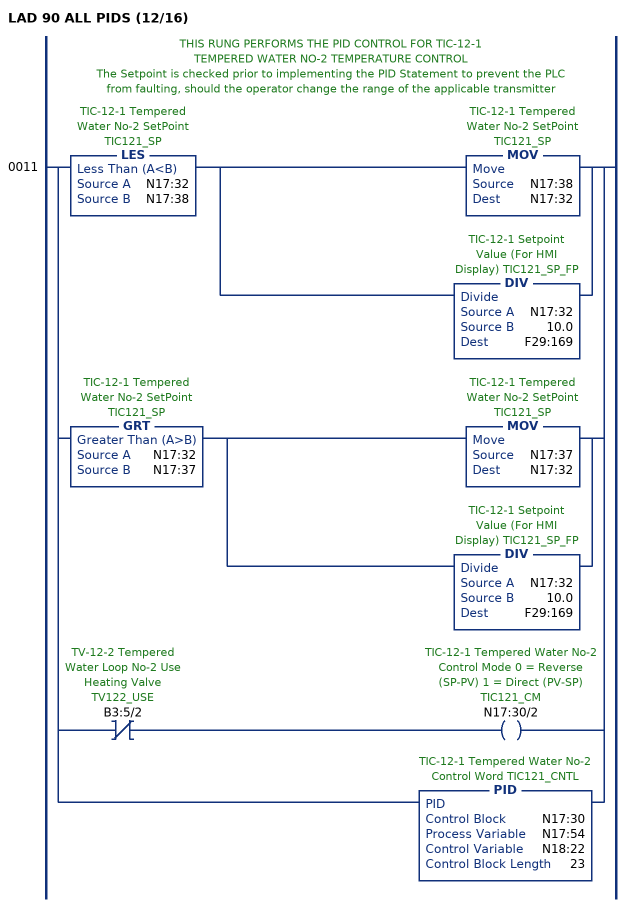
% Rung: 11 %
% THIS RUNG PERFORMS THE PID CONTROL FOR TIC-12-1
% TEMPERED WATER NO-2 TEMPERATURE CONTROL
% The Setpoint is checked prior to implementing the PID Statement to prevent the PLC
% from faulting, should the operator change the range of the applicable transmitter %
SOR BST LES N17:32 N17:38 BST MOV N17:38 N17:32 NXB DIV N17:32 10.0 F29:169 BND NXB GRT N17:32 N17:37 BST MOV N17:37 N17:32 NXB DIV N17:32 10.0 F29:169 BND NXB XIO B3:5/2 OTE N17:30/2 NXB PID N17:30 N17:54 N18:22 23 BND EOR
%   N17:32  TIC121_SP  "TIC-12-1 Tempered Water No-2 SetPoint" %
%   N17:38  TIC121_SMIN  "TIC-12-1 Tempered Water No-2 Setpoint Minimum" %
%   F29:169  TIC121_SP_FP  "TIC-12-1 Setpoint Value (For HMI Display)" %
%   N17:37  TIC121_SMAX  "TIC-12-1 Tempered Water No-2 Setpoint Maximum" %
%   B3:5/2  TV122_USE  "TV-12-2 Tempered Water Loop No-2 Use Heating Valve" %
%   N17:30/2  TIC121_CM  "TIC-12-1 Tempered Water No-2 Control Mode 0 = Reverse (SP-PV) 1 = Direct (PV-SP)" %
%   N17:30  TIC121_CNTL  "TIC-12-1 Tempered Water No-2 Control Word" %
%   N17:54  TIC121_IN  "TIC-12-1 Tempered Water No-2 Scaled Input" %
%   N18:22  TIC121_OUT1  "TIC-12-1 Tempered Water No-2 PID Output Value" %

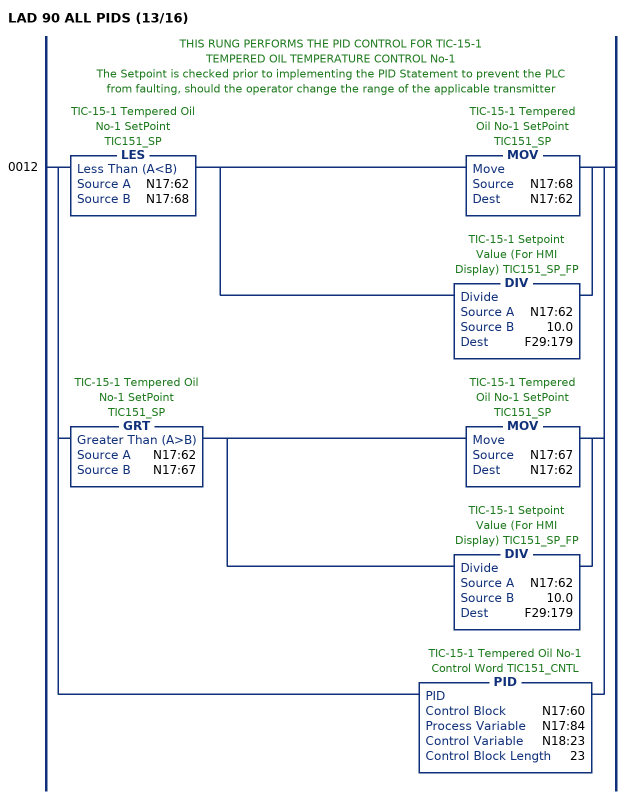
% Rung: 12 %
% THIS RUNG PERFORMS THE PID CONTROL FOR TIC-15-1
% TEMPERED OIL TEMPERATURE CONTROL No-1
% The Setpoint is checked prior to implementing the PID Statement to prevent the PLC
% from faulting, should the operator change the range of the applicable transmitter %
SOR BST LES N17:62 N17:68 BST MOV N17:68 N17:62 NXB DIV N17:62 10.0 F29:179 BND NXB GRT N17:62 N17:67 BST MOV N17:67 N17:62 NXB DIV N17:62 10.0 F29:179 BND NXB PID N17:60 N17:84 N18:23 23 BND EOR
%   N17:62  TIC151_SP  "TIC-15-1 Tempered Oil No-1 SetPoint" %
%   N17:68  TIC151_SMIN  "TIC-15-1 Tempered Oil No-1 Setpoint Minimum" %
%   F29:179  TIC151_SP_FP  "TIC-15-1 Setpoint Value (For HMI Display)" %
%   N17:67  TIC151_SMAX  "TIC-15-1 Tempered Oil No-1 Setpoint Maximum" %
%   N17:60  TIC151_CNTL  "TIC-15-1 Tempered Oil No-1 Control Word" %
%   N17:84  TIC151_IN  "TIC-15-1 Tempered Oil No-1 Scaled Input" %
%   N18:23  TIC151_OUT1  "TIC-15-1 Tempered Oil No-1 PID Output Value" %

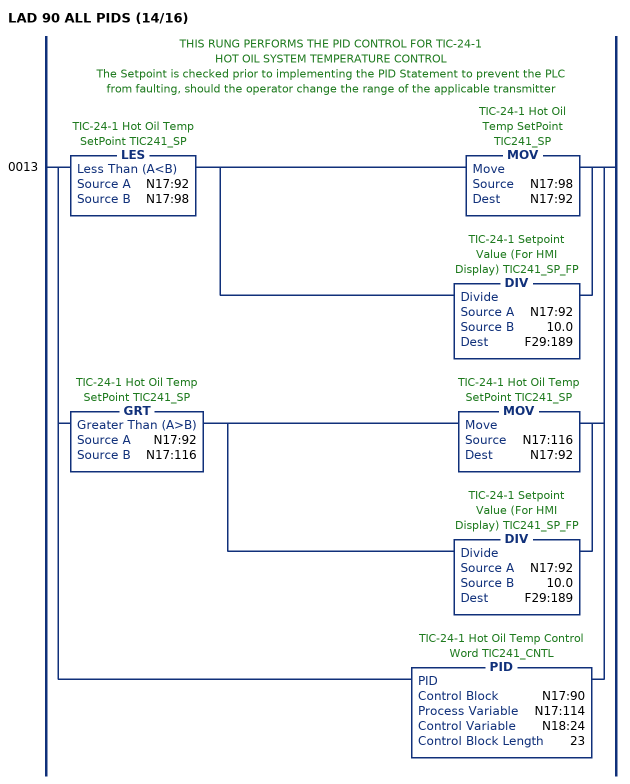
% Rung: 13 %
% THIS RUNG PERFORMS THE PID CONTROL FOR TIC-24-1
% HOT OIL SYSTEM TEMPERATURE CONTROL
% The Setpoint is checked prior to implementing the PID Statement to prevent the PLC
% from faulting, should the operator change the range of the applicable transmitter %
SOR BST LES N17:92 N17:98 BST MOV N17:98 N17:92 NXB DIV N17:92 10.0 F29:189 BND NXB GRT N17:92 N17:116 BST MOV N17:116 N17:92 NXB DIV N17:92 10.0 F29:189 BND NXB PID N17:90 N17:114 N18:24 23 BND EOR
%   N17:92  TIC241_SP  "TIC-24-1 Hot Oil Temp SetPoint" %
%   N17:98  TIC241_SMIN  "TIC-24-1 Hot Oil Temp Setpoint Minimum" %
%   F29:189  TIC241_SP_FP  "TIC-24-1 Setpoint Value (For HMI Display)" %
%   N17:116  TIC241_OPER_SPMAX  "TIC-24-1 Operating Setpoint Max" %
%   N17:90  TIC241_CNTL  "TIC-24-1 Hot Oil Temp Control Word" %
%   N17:114  TIC241_IN  "TIC-24-1 Hot Oil Temp Scaled Input" %
%   N18:24  TIC241_OUT1  "TIC-24-1 Hot Oil Temp PID Output Value" %

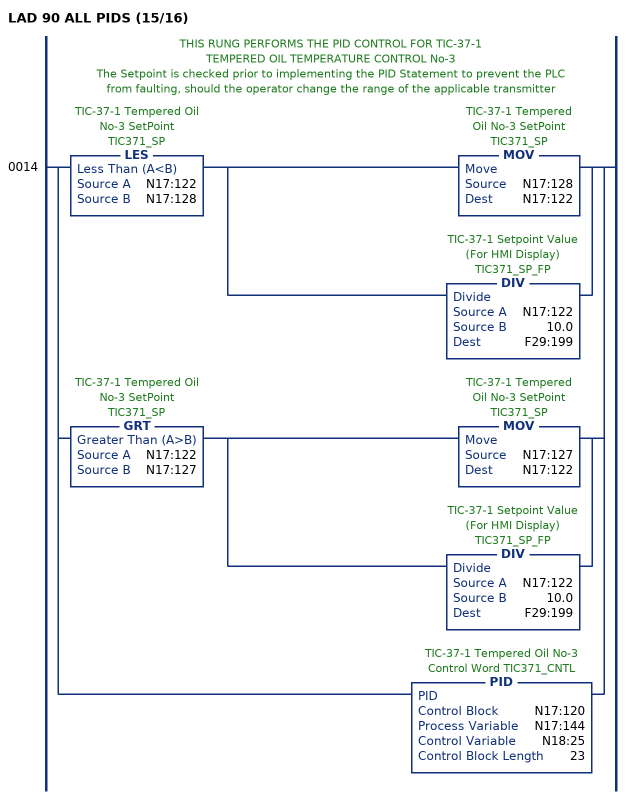
% Rung: 14 %
% THIS RUNG PERFORMS THE PID CONTROL FOR TIC-37-1
% TEMPERED OIL TEMPERATURE CONTROL No-3
% The Setpoint is checked prior to implementing the PID Statement to prevent the PLC
% from faulting, should the operator change the range of the applicable transmitter %
SOR BST LES N17:122 N17:128 BST MOV N17:128 N17:122 NXB DIV N17:122 10.0 F29:199 BND NXB GRT N17:122 N17:127 BST MOV N17:127 N17:122 NXB DIV N17:122 10.0 F29:199 BND NXB PID N17:120 N17:144 N18:25 23 BND EOR
%   N17:122  TIC371_SP  "TIC-37-1 Tempered Oil No-3 SetPoint" %
%   N17:128  TIC371_SMIN  "TIC-37-1 Tempered Oil No-3 Setpoint Minimum" %
%   F29:199  TIC371_SP_FP  "TIC-37-1 Setpoint Value (For HMI Display)" %
%   N17:127  TIC371_SMAX  "TIC-37-1 Tempered Oil No-3 Setpoint Maximum" %
%   N17:120  TIC371_CNTL  "TIC-37-1 Tempered Oil No-3 Control Word" %
%   N17:144  TIC371_IN  "TIC-37-1 Tempered Oil No-3 Scaled Input" %
%   N18:25  TIC371_OUT1  "TIC-37-1 Tempered Oil No-3 PID Output Value" %

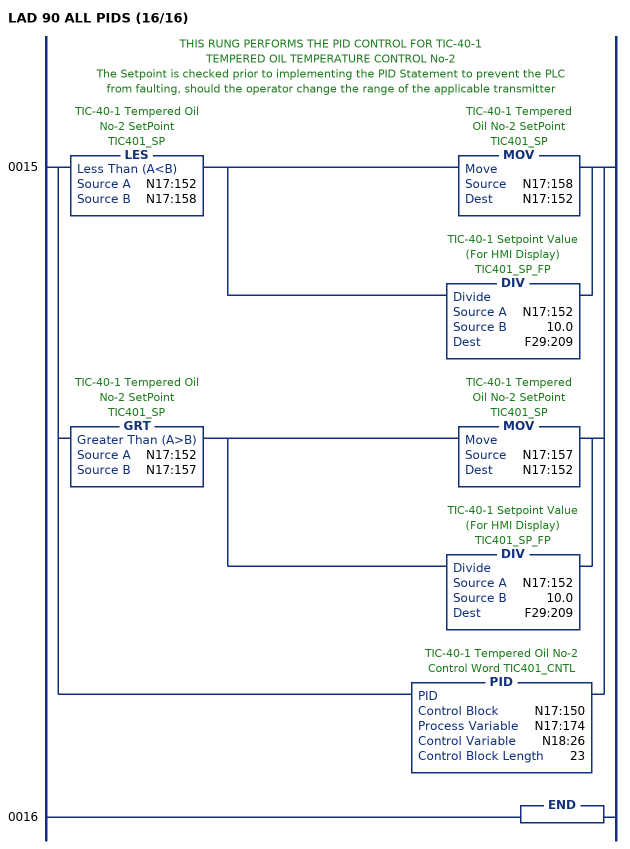
% Rung: 15 %
% THIS RUNG PERFORMS THE PID CONTROL FOR TIC-40-1
% TEMPERED OIL TEMPERATURE CONTROL No-2
% The Setpoint is checked prior to implementing the PID Statement to prevent the PLC
% from faulting, should the operator change the range of the applicable transmitter %
SOR BST LES N17:152 N17:158 BST MOV N17:158 N17:152 NXB DIV N17:152 10.0 F29:209 BND NXB GRT N17:152 N17:157 BST MOV N17:157 N17:152 NXB DIV N17:152 10.0 F29:209 BND NXB PID N17:150 N17:174 N18:26 23 BND EOR
%   N17:152  TIC401_SP  "TIC-40-1 Tempered Oil No-2 SetPoint" %
%   N17:158  TIC401_SMIN  "TIC-40-1 Tempered Oil No-2 Setpoint Minimum" %
%   F29:209  TIC401_SP_FP  "TIC-40-1 Setpoint Value (For HMI Display)" %
%   N17:157  TIC401_SMAX  "TIC-40-1 Tempered Oil No-2 Setpoint Maximum" %
%   N17:150  TIC401_CNTL  "TIC-40-1 Tempered Oil No-2 Control Word" %
%   N17:174  TIC401_IN  "TIC-40-1 Tempered Oil No-2 Scaled Input" %
%   N18:26  TIC401_OUT1  "TIC-40-1 Tempered Oil No-2 PID Output Value" %
% Rung: 16 %
SOR END EOR

LADDER 101 "FIC-21-1"    % Feed Flow No-1 PID Controls %
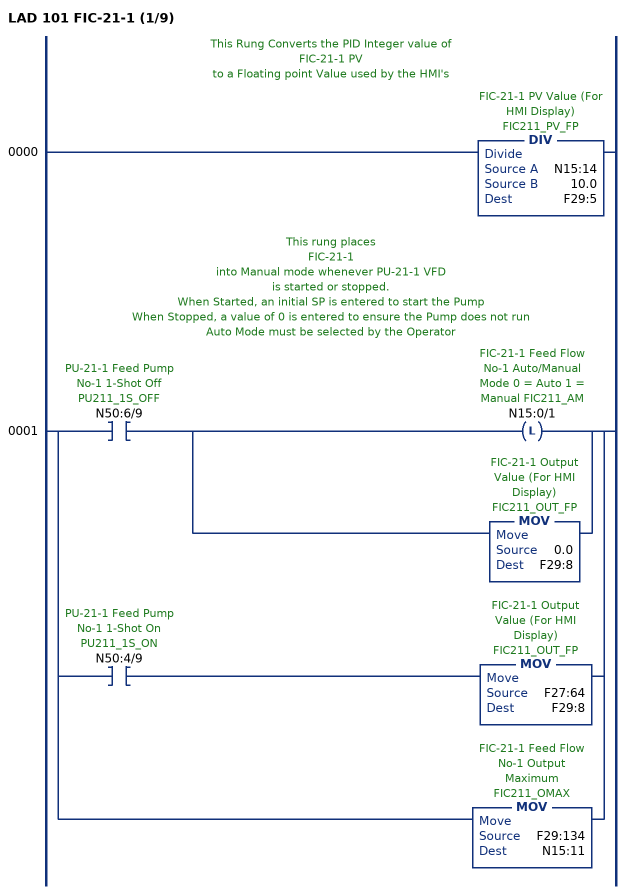
% Rung: 0 %
% This Rung Converts the PID Integer value of
% FIC-21-1 PV
% to a Floating point Value used by the HMI's %
SOR DIV N15:14 10.0 F29:5 EOR
%   N15:14  FIC211_PV  "FIC-21-1 Feed Flow No-1 Scaled Process Variable" %
%   F29:5  FIC211_PV_FP  "FIC-21-1 PV Value (For HMI Display)" %
% Rung: 1 %
% This rung places
% FIC-21-1
% into Manual mode whenever PU-21-1 VFD
% is started or stopped.
% When Started, an initial SP is entered to start the Pump
% When Stopped, a value of 0 is entered to ensure the Pump does not run
% Auto Mode must be selected by the Operator %
SOR BST XIC N50:6/9 BST OTL N15:0/1 NXB MOV 0.0 F29:8 BND NXB XIC N50:4/9 MOV F27:64 F29:8 NXB MOV F29:134 N15:11 BND EOR
%   N50:6/9  PU211_1S_OFF  "PU-21-1 Feed Pump No-1 1-Shot Off" %
%   N15:0/1  FIC211_AM  "FIC-21-1 Feed Flow No-1 Auto/Manual Mode 0 = Auto 1 = Manual" %
%   F29:8  FIC211_OUT_FP  "FIC-21-1 Output Value (For HMI Display)" %
%   N50:4/9  PU211_1S_ON  "PU-21-1 Feed Pump No-1 1-Shot On" %
%   F27:64  SIC211_INIT_SP  "SIC-21-1 Initial Speed Setpoint (Hz)" %
%   F29:134  SIC211_MAX  "SIC-21-1 PU-21-1 Feed Pump No-1 Freq at 100% Value (For HMI Display)" %
%   N15:11  FIC211_OMAX  "FIC-21-1 Feed Flow No-1 Output Maximum" %

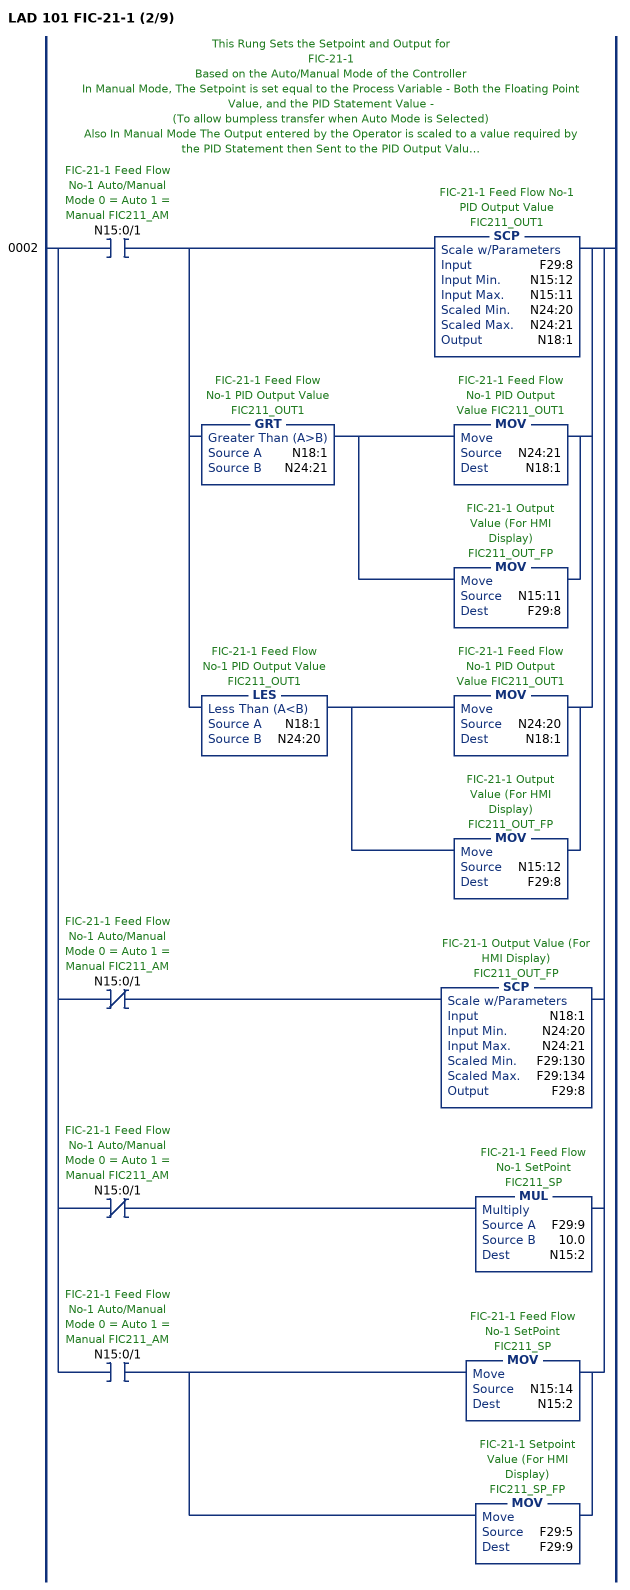
% Rung: 2 %
% This Rung Sets the Setpoint and Output for
% FIC-21-1
% Based on the Auto/Manual Mode of the Controller
% In Manual Mode, The Setpoint is set equal to the Process Variable - Both the Floating Point Value, and the PID Statement Value -
% (To allow bumpless transfer when Auto Mode is Selected)
% Also In Manual Mode The Output entered by the Operator is scaled to a value required by the PID Statement then Sent to the PID Output Value
% 
% In Auto Mode, The Setpoint is Entered by the Operator from Any HMI terminal, Multiplied by 10, and placed in the PID Statement's Setpoint Location
% Also In Auto Mode, the Output (used by the Operator) is set equal to the actual value of the pID statement
% (To allow bumpless transfer when Manual Mode is Selected) %
SOR BST XIC N15:0/1 BST SCP F29:8 N15:12 N15:11 N24:20 N24:21 N18:1 NXB GRT N18:1 N24:21 BST MOV N24:21 N18:1 NXB MOV N15:11 F29:8 BND NXB LES N18:1 N24:20 BST MOV N24:20 N18:1 NXB MOV N15:12 F29:8 BND BND NXB XIO N15:0/1 SCP N18:1 N24:20 N24:21 F29:130 F29:134 F29:8 NXB XIO N15:0/1 MUL F29:9 10.0 N15:2 NXB XIC N15:0/1 BST MOV N15:14 N15:2 NXB MOV F29:5 F29:9 BND BND EOR
%   N15:0/1  FIC211_AM  "FIC-21-1 Feed Flow No-1 Auto/Manual Mode 0 = Auto 1 = Manual" %
%   F29:8  FIC211_OUT_FP  "FIC-21-1 Output Value (For HMI Display)" %
%   N15:12  FIC211_OMIN  "FIC-21-1 Feed Flow No-1 Output Minimum" %
%   N15:11  FIC211_OMAX  "FIC-21-1 Feed Flow No-1 Output Maximum" %
%   N24:20  PID_MIN  "PID Statement Minimum Value" %
%   N24:21  PID_MAX  "PID Statement Maximum Value" %
%   N18:1  FIC211_OUT1  "FIC-21-1 Feed Flow No-1 PID Output Value" %
%   F29:130  SIC211_MIN  "SIC-21-1 PU-21-1 Feed Pump No-1 Speed 0% Value (For HMI Display)" %
%   F29:134  SIC211_MAX  "SIC-21-1 PU-21-1 Feed Pump No-1 Freq at 100% Value (For HMI Display)" %
%   F29:9  FIC211_SP_FP  "FIC-21-1 Setpoint Value (For HMI Display)" %
%   N15:2  FIC211_SP  "FIC-21-1 Feed Flow No-1 SetPoint" %
%   N15:14  FIC211_PV  "FIC-21-1 Feed Flow No-1 Scaled Process Variable" %
%   F29:5  FIC211_PV_FP  "FIC-21-1 PV Value (For HMI Display)" %

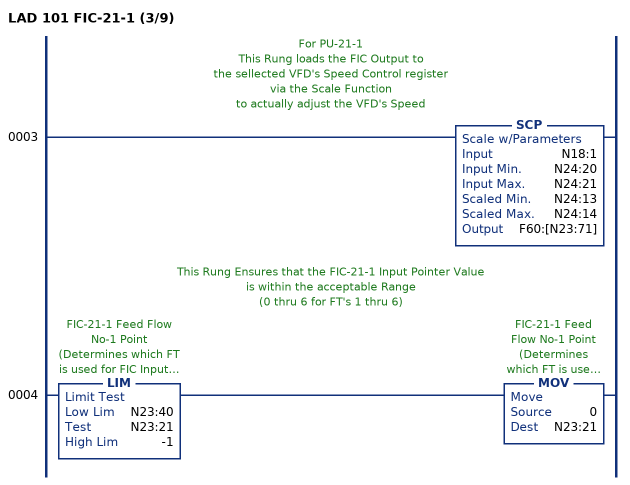
% Rung: 3 %
% For PU-21-1
% This Rung loads the FIC Output to
% the sellected VFD's Speed Control register
% via the Scale Function
% to actually adjust the VFD's Speed %
SOR SCP N18:1 N24:20 N24:21 N24:13 N24:14 F60:[N23:71] EOR
%   N18:1  FIC211_OUT1  "FIC-21-1 Feed Flow No-1 PID Output Value" %
%   N24:20  PID_MIN  "PID Statement Minimum Value" %
%   N24:21  PID_MAX  "PID Statement Maximum Value" %
%   N24:13  AO_MIN_OE4  "Analog Output Minimum Value Generates 4 mA DC (To OE4 AO Module)" %
%   N24:14  AO_MAX_OE4  "Analog Output Maximum Value Generates 20 mA DC (To OE4 AO Module)" %
%   N23:71  FIC211_OUT_PTR  "FIC-21-1 Feed Flow No-1 Output Pointer Determines which VFD is controled by FIC" %
% Rung: 4 %
% This Rung Ensures that the FIC-21-1 Input Pointer Value
% is within the acceptable Range
% (0 thru 6 for FT's 1 thru 6) %
SOR LIM N23:40 N23:21 -1 MOV 0 N23:21 EOR
%   N23:40  MAX_FT_ALLOWED_1  "Maximum Number of FTs Available Plus 1" %
%   N23:21  FIC211_IN_PTR  "FIC-21-1 Feed Flow No-1 Point (Determines which FT is used for FIC Input)" %

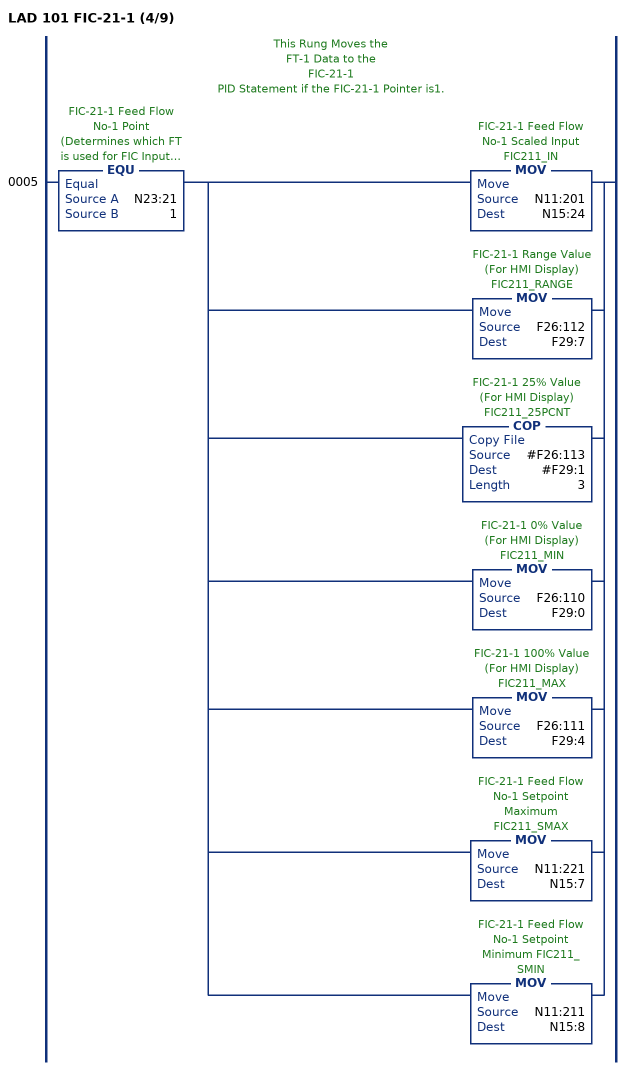
% Rung: 5 %
% This Rung Moves the
% FT-1 Data to the
% FIC-21-1
% PID Statement if the FIC-21-1 Pointer is1. %
SOR EQU N23:21 1 BST MOV N11:201 N15:24 NXB MOV F26:112 F29:7 NXB COP #F26:113 #F29:1 3 NXB MOV F26:110 F29:0 NXB MOV F26:111 F29:4 NXB MOV N11:221 N15:7 NXB MOV N11:211 N15:8 BND EOR
%   N23:21  FIC211_IN_PTR  "FIC-21-1 Feed Flow No-1 Point (Determines which FT is used for FIC Input)" %
%   N11:201  FT01_PID_IN  "FT-1 Flow Transmitter No-1 PID Statement Input Value" %
%   N15:24  FIC211_IN  "FIC-21-1 Feed Flow No-1 Scaled Input" %
%   F26:112  FT01_RANGE  "FT-1 Range Value (Max-Min)" %
%   F29:7  FIC211_RANGE  "FIC-21-1 Range Value (For HMI Display)" %
%   F26:113  FT01_25PCNT_VALUE  "FT-1 25% Range Value For HMI Display" %
%   F29:1  FIC211_25PCNT  "FIC-21-1 25% Value (For HMI Display)" %
%   F26:110  FT01_MIN  "FT-1 Minimum Value" %
%   F29:0  FIC211_MIN  "FIC-21-1 0% Value (For HMI Display)" %
%   F26:111  FT01_MAX  "FT-1 Maximum Value" %
%   F29:4  FIC211_MAX  "FIC-21-1 100% Value (For HMI Display)" %
%   N11:221  FT01_PID_MAX  "FT-1 Flow Transmitter No-1 PID Statement Maximum Input Value" %
%   N15:7  FIC211_SMAX  "FIC-21-1 Feed Flow No-1 Setpoint Maximum" %
%   N11:211  FT01_PID_MIN  "FT-1 Flow Transmitter No-1 PID Statement Minimum Input Value" %
%   N15:8  FIC211_SMIN  "FIC-21-1 Feed Flow No-1 Setpoint Minimum" %

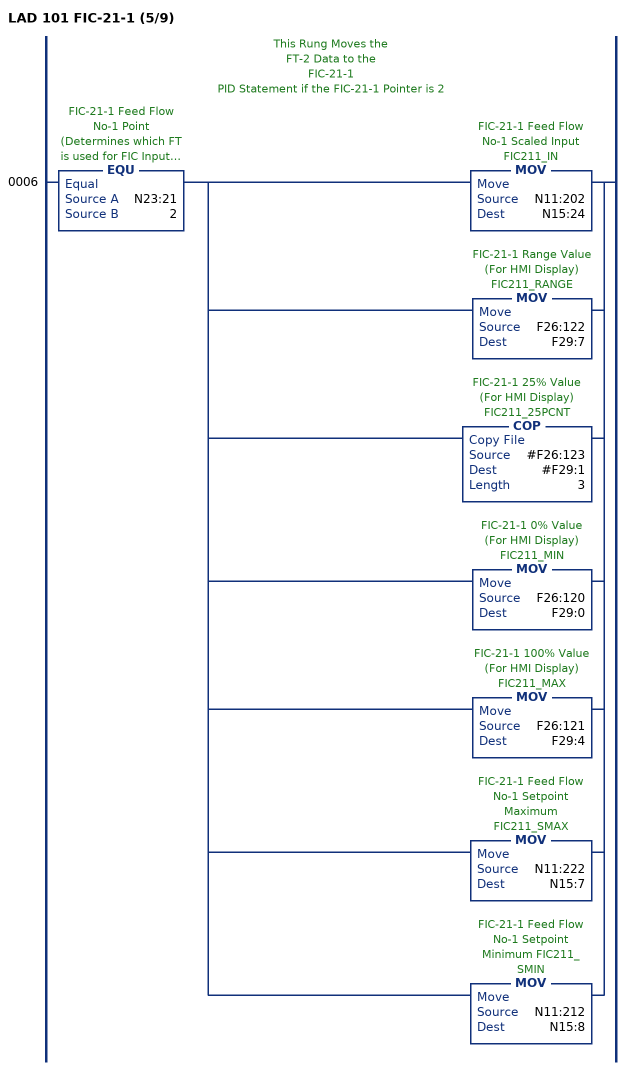
% Rung: 6 %
% This Rung Moves the
% FT-2 Data to the
% FIC-21-1
% PID Statement if the FIC-21-1 Pointer is 2 %
SOR EQU N23:21 2 BST MOV N11:202 N15:24 NXB MOV F26:122 F29:7 NXB COP #F26:123 #F29:1 3 NXB MOV F26:120 F29:0 NXB MOV F26:121 F29:4 NXB MOV N11:222 N15:7 NXB MOV N11:212 N15:8 BND EOR
%   N23:21  FIC211_IN_PTR  "FIC-21-1 Feed Flow No-1 Point (Determines which FT is used for FIC Input)" %
%   N11:202  FT02_PID_IN  "FT-2 Flow Transmitter No-2 PID Statement Input Value" %
%   N15:24  FIC211_IN  "FIC-21-1 Feed Flow No-1 Scaled Input" %
%   F26:122  FT02_RANGE  "FT-2 Range Value (Max-Min)" %
%   F29:7  FIC211_RANGE  "FIC-21-1 Range Value (For HMI Display)" %
%   F26:123  FT02_25PCNT_VALUE  "FT-2 25% Range Value For HMI Display" %
%   F29:1  FIC211_25PCNT  "FIC-21-1 25% Value (For HMI Display)" %
%   F26:120  FT02_MIN  "FT-2 Minimum Value" %
%   F29:0  FIC211_MIN  "FIC-21-1 0% Value (For HMI Display)" %
%   F26:121  FT02_MAX  "FT-2 Maximum Value" %
%   F29:4  FIC211_MAX  "FIC-21-1 100% Value (For HMI Display)" %
%   N11:222  FT02_PID_MAX  "FT-2 Flow Transmitter No-2 PID Statement Maximum Input Value" %
%   N15:7  FIC211_SMAX  "FIC-21-1 Feed Flow No-1 Setpoint Maximum" %
%   N11:212  FT02_PID_MIN  "FT-2 Flow Transmitter No-2 PID Statement Minimum Input Value" %
%   N15:8  FIC211_SMIN  "FIC-21-1 Feed Flow No-1 Setpoint Minimum" %

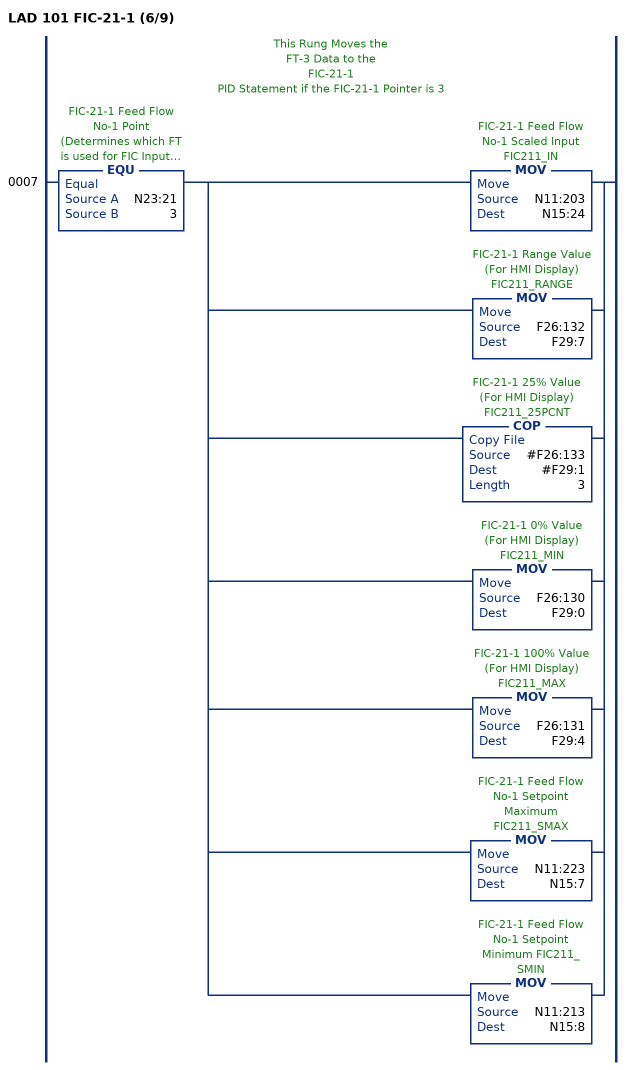
% Rung: 7 %
% This Rung Moves the
% FT-3 Data to the
% FIC-21-1
% PID Statement if the FIC-21-1 Pointer is 3 %
SOR EQU N23:21 3 BST MOV N11:203 N15:24 NXB MOV F26:132 F29:7 NXB COP #F26:133 #F29:1 3 NXB MOV F26:130 F29:0 NXB MOV F26:131 F29:4 NXB MOV N11:223 N15:7 NXB MOV N11:213 N15:8 BND EOR
%   N23:21  FIC211_IN_PTR  "FIC-21-1 Feed Flow No-1 Point (Determines which FT is used for FIC Input)" %
%   N11:203  FT03_PID_IN  "FT-3 Flow Transmitter No-3 PID Statement Input Value" %
%   N15:24  FIC211_IN  "FIC-21-1 Feed Flow No-1 Scaled Input" %
%   F26:132  FT03_RANGE  "FT-3 Range Value (Max-Min)" %
%   F29:7  FIC211_RANGE  "FIC-21-1 Range Value (For HMI Display)" %
%   F26:133  FT03_25PCNT_VALUE  "FT-3 25% Range Value For HMI Display" %
%   F29:1  FIC211_25PCNT  "FIC-21-1 25% Value (For HMI Display)" %
%   F26:130  FT03_MIN  "FT-3 Minimum Value" %
%   F29:0  FIC211_MIN  "FIC-21-1 0% Value (For HMI Display)" %
%   F26:131  FT03_MAX  "FT-3 Maximum Value" %
%   F29:4  FIC211_MAX  "FIC-21-1 100% Value (For HMI Display)" %
%   N11:223  FT03_PID_MAX  "FT-3 Flow Transmitter No-3 PID Statement Maximum Input Value" %
%   N15:7  FIC211_SMAX  "FIC-21-1 Feed Flow No-1 Setpoint Maximum" %
%   N11:213  FT03_PID_MIN  "FT-3 Flow Transmitter No-3 PID Statement Minimum Input Value" %
%   N15:8  FIC211_SMIN  "FIC-21-1 Feed Flow No-1 Setpoint Minimum" %

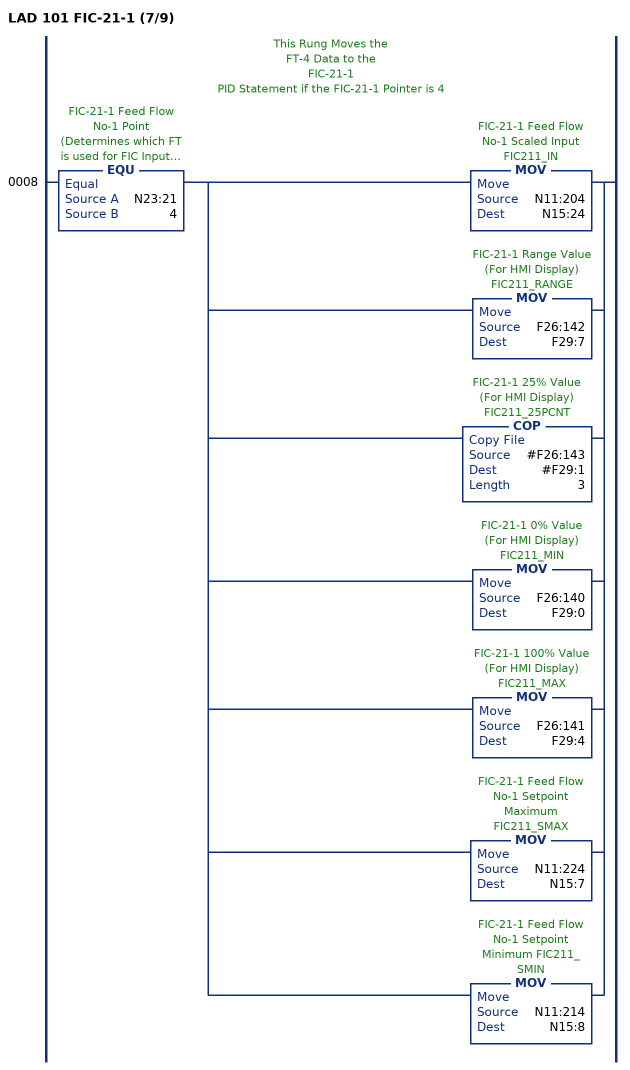
% Rung: 8 %
% This Rung Moves the
% FT-4 Data to the
% FIC-21-1
% PID Statement if the FIC-21-1 Pointer is 4 %
SOR EQU N23:21 4 BST MOV N11:204 N15:24 NXB MOV F26:142 F29:7 NXB COP #F26:143 #F29:1 3 NXB MOV F26:140 F29:0 NXB MOV F26:141 F29:4 NXB MOV N11:224 N15:7 NXB MOV N11:214 N15:8 BND EOR
%   N23:21  FIC211_IN_PTR  "FIC-21-1 Feed Flow No-1 Point (Determines which FT is used for FIC Input)" %
%   N11:204  FT04_PID_IN  "FT-4 Flow Transmitter No-4 PID Statement Input Value" %
%   N15:24  FIC211_IN  "FIC-21-1 Feed Flow No-1 Scaled Input" %
%   F26:142  FT04_RANGE  "FT-4 Range Value (Max-Min)" %
%   F29:7  FIC211_RANGE  "FIC-21-1 Range Value (For HMI Display)" %
%   F26:143  FT04_25PCNT_VALUE  "FT-4 25% Range Value For HMI Display" %
%   F29:1  FIC211_25PCNT  "FIC-21-1 25% Value (For HMI Display)" %
%   F26:140  FT04_MIN  "FT-4 Minimum Value" %
%   F29:0  FIC211_MIN  "FIC-21-1 0% Value (For HMI Display)" %
%   F26:141  FT04_MAX  "FT-4 Maximum Value" %
%   F29:4  FIC211_MAX  "FIC-21-1 100% Value (For HMI Display)" %
%   N11:224  FT04_PID_MAX  "FT-4 Flow Transmitter No-4 PID Statement Maximum Input Value" %
%   N15:7  FIC211_SMAX  "FIC-21-1 Feed Flow No-1 Setpoint Maximum" %
%   N11:214  FT04_PID_MIN  "FT-4 Flow Transmitter No-4 PID Statement Minimum Input Value" %
%   N15:8  FIC211_SMIN  "FIC-21-1 Feed Flow No-1 Setpoint Minimum" %

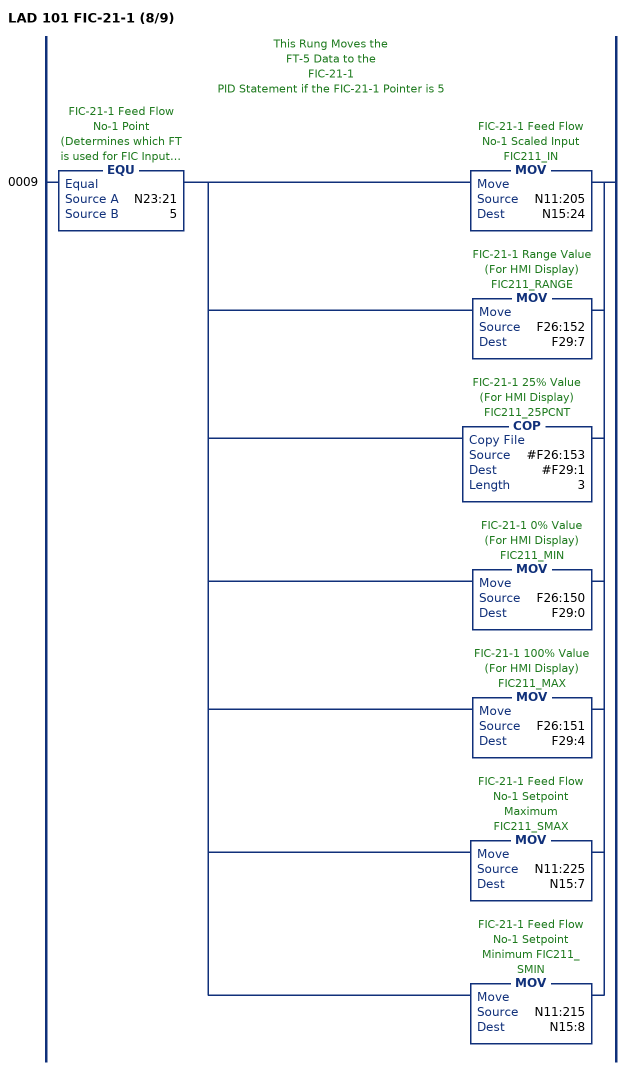
% Rung: 9 %
% This Rung Moves the
% FT-5 Data to the
% FIC-21-1
% PID Statement if the FIC-21-1 Pointer is 5 %
SOR EQU N23:21 5 BST MOV N11:205 N15:24 NXB MOV F26:152 F29:7 NXB COP #F26:153 #F29:1 3 NXB MOV F26:150 F29:0 NXB MOV F26:151 F29:4 NXB MOV N11:225 N15:7 NXB MOV N11:215 N15:8 BND EOR
%   N23:21  FIC211_IN_PTR  "FIC-21-1 Feed Flow No-1 Point (Determines which FT is used for FIC Input)" %
%   N11:205  FT05_PID_IN  "FT-5 Flow Transmitter No-5 PID Statement Input Value" %
%   N15:24  FIC211_IN  "FIC-21-1 Feed Flow No-1 Scaled Input" %
%   F26:152  FT05_RANGE  "FT-5 Range Value (Max-Min)" %
%   F29:7  FIC211_RANGE  "FIC-21-1 Range Value (For HMI Display)" %
%   F26:153  FT05_25PCNT_VALUE  "FT-5 25% Range Value For HMI Display" %
%   F29:1  FIC211_25PCNT  "FIC-21-1 25% Value (For HMI Display)" %
%   F26:150  FT05_MIN  "FT-5 Minimum Value" %
%   F29:0  FIC211_MIN  "FIC-21-1 0% Value (For HMI Display)" %
%   F26:151  FT05_MAX  "FT-5 Maximum Value" %
%   F29:4  FIC211_MAX  "FIC-21-1 100% Value (For HMI Display)" %
%   N11:225  FT05_PID_MAX  "FT-5 Flow Transmitter No-5 PID Statement Maximum Input Value" %
%   N15:7  FIC211_SMAX  "FIC-21-1 Feed Flow No-1 Setpoint Maximum" %
%   N11:215  FT05_PID_MIN  "FT-5 Flow Transmitter No-5 PID Statement Minimum Input Value" %
%   N15:8  FIC211_SMIN  "FIC-21-1 Feed Flow No-1 Setpoint Minimum" %

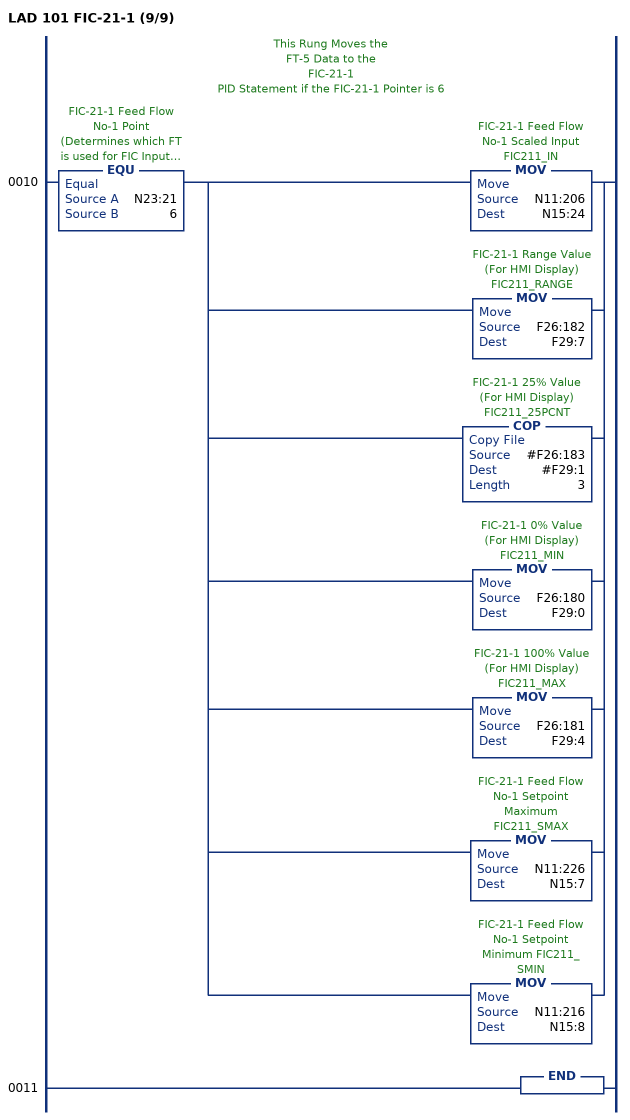
% Rung: 10 %
% This Rung Moves the
% FT-5 Data to the
% FIC-21-1
% PID Statement if the FIC-21-1 Pointer is 6 %
SOR EQU N23:21 6 BST MOV N11:206 N15:24 NXB MOV F26:182 F29:7 NXB COP #F26:183 #F29:1 3 NXB MOV F26:180 F29:0 NXB MOV F26:181 F29:4 NXB MOV N11:226 N15:7 NXB MOV N11:216 N15:8 BND EOR
%   N23:21  FIC211_IN_PTR  "FIC-21-1 Feed Flow No-1 Point (Determines which FT is used for FIC Input)" %
%   N11:206  FT06_PID_IN  "FT-6 Flow Transmitter No-6 PID Statement Input Value" %
%   N15:24  FIC211_IN  "FIC-21-1 Feed Flow No-1 Scaled Input" %
%   F26:182  FT06_RANGE  "FT-6 Range Value (Max-Min)" %
%   F29:7  FIC211_RANGE  "FIC-21-1 Range Value (For HMI Display)" %
%   F26:183  FT06_25PCNT_VALUE  "FT-6 25% Range Value For HMI Display" %
%   F29:1  FIC211_25PCNT  "FIC-21-1 25% Value (For HMI Display)" %
%   F26:180  FT06_MIN  "FT-6 Minimum Value" %
%   F29:0  FIC211_MIN  "FIC-21-1 0% Value (For HMI Display)" %
%   F26:181  FT06_MAX  "FT-6 Maximum Value" %
%   F29:4  FIC211_MAX  "FIC-21-1 100% Value (For HMI Display)" %
%   N11:226  FT06_PID_MAX  "FT-6 Flow Transmitter No-6 PID Statement Maximum Input Value" %
%   N15:7  FIC211_SMAX  "FIC-21-1 Feed Flow No-1 Setpoint Maximum" %
%   N11:216  FT06_PID_MIN  "FT-6 Flow Transmitter No-6 PID Statement Minimum Input Value" %
%   N15:8  FIC211_SMIN  "FIC-21-1 Feed Flow No-1 Setpoint Minimum" %
% Rung: 11 %
SOR END EOR

LADDER 102 "FIC-21-2"    % Feed Flow No-2 PID Controls %
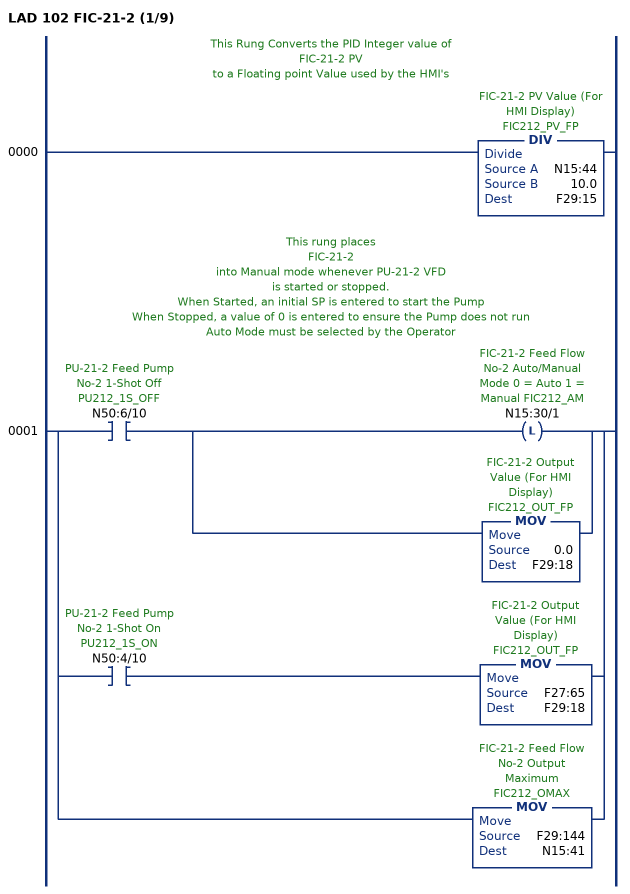
% Rung: 0 %
% This Rung Converts the PID Integer value of
% FIC-21-2 PV
% to a Floating point Value used by the HMI's %
SOR DIV N15:44 10.0 F29:15 EOR
%   N15:44  FIC212_PV  "FIC-21-2 Feed Flow No-2 Scaled Process Variable" %
%   F29:15  FIC212_PV_FP  "FIC-21-2 PV Value (For HMI Display)" %
% Rung: 1 %
% This rung places
% FIC-21-2
% into Manual mode whenever PU-21-2 VFD
% is started or stopped.
% When Started, an initial SP is entered to start the Pump
% When Stopped, a value of 0 is entered to ensure the Pump does not run
% Auto Mode must be selected by the Operator %
SOR BST XIC N50:6/10 BST OTL N15:30/1 NXB MOV 0.0 F29:18 BND NXB XIC N50:4/10 MOV F27:65 F29:18 NXB MOV F29:144 N15:41 BND EOR
%   N50:6/10  PU212_1S_OFF  "PU-21-2 Feed Pump No-2 1-Shot Off" %
%   N15:30/1  FIC212_AM  "FIC-21-2 Feed Flow No-2 Auto/Manual Mode 0 = Auto 1 = Manual" %
%   F29:18  FIC212_OUT_FP  "FIC-21-2 Output Value (For HMI Display)" %
%   N50:4/10  PU212_1S_ON  "PU-21-2 Feed Pump No-2 1-Shot On" %
%   F27:65  SIC212_INIT_SP  "SIC-21-2 Initial Speed Setpoint (Hz)" %
%   F29:144  SIC212_MAX  "SIC-21-2 PU-21-2 Feed Pump No-2 Freq at 100% Value (For HMI Display)" %
%   N15:41  FIC212_OMAX  "FIC-21-2 Feed Flow No-2 Output Maximum" %

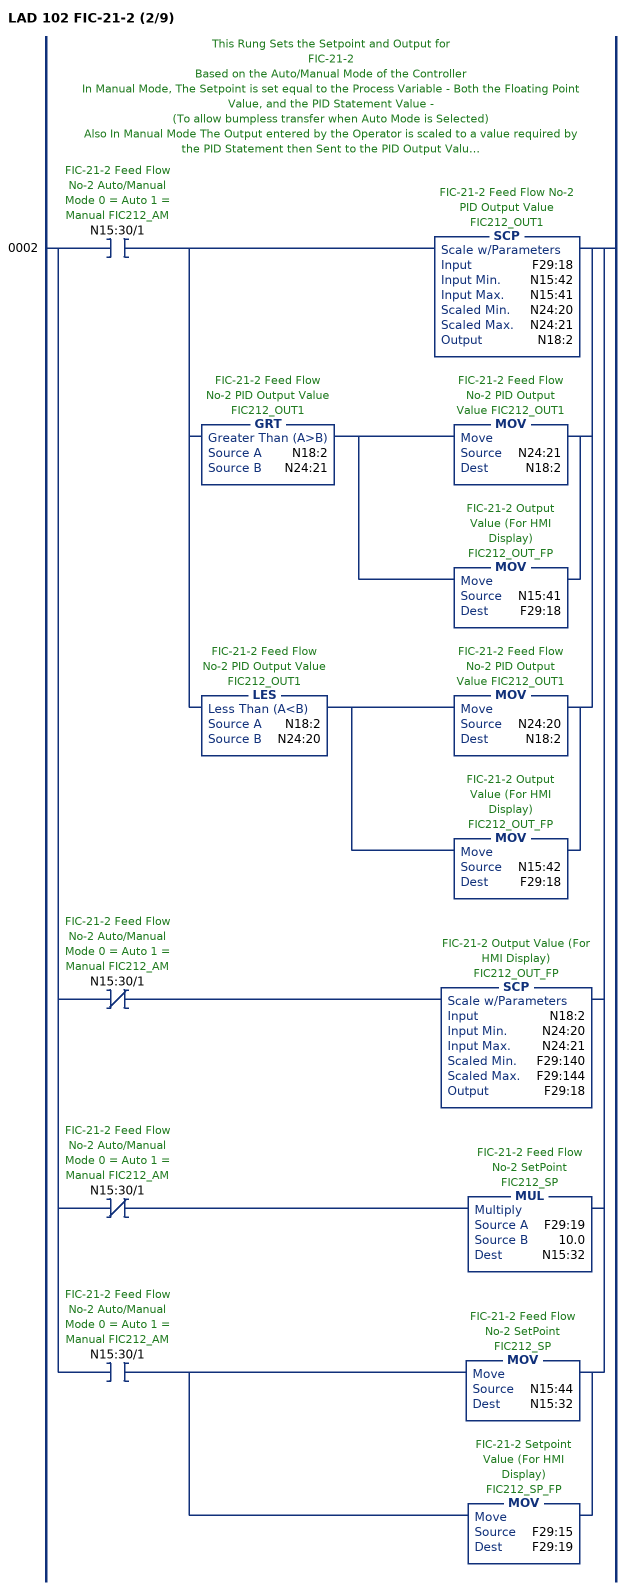
% Rung: 2 %
% This Rung Sets the Setpoint and Output for
% FIC-21-2
% Based on the Auto/Manual Mode of the Controller
% In Manual Mode, The Setpoint is set equal to the Process Variable - Both the Floating Point Value, and the PID Statement Value -
% (To allow bumpless transfer when Auto Mode is Selected)
% Also In Manual Mode The Output entered by the Operator is scaled to a value required by the PID Statement then Sent to the PID Output Value
% 
% In Auto Mode, The Setpoint is Entered by the Operator from Any HMI terminal, Multiplied by 10, and placed in the PID Statement's Setpoint Location
% Also In Auto Mode, the Output (used by the Operator) is set equal to the actual value of the pID statement
% (To allow bumpless transfer when Manual Mode is Selected) %
SOR BST XIC N15:30/1 BST SCP F29:18 N15:42 N15:41 N24:20 N24:21 N18:2 NXB GRT N18:2 N24:21 BST MOV N24:21 N18:2 NXB MOV N15:41 F29:18 BND NXB LES N18:2 N24:20 BST MOV N24:20 N18:2 NXB MOV N15:42 F29:18 BND BND NXB XIO N15:30/1 SCP N18:2 N24:20 N24:21 F29:140 F29:144 F29:18 NXB XIO N15:30/1 MUL F29:19 10.0 N15:32 NXB XIC N15:30/1 BST MOV N15:44 N15:32 NXB MOV F29:15 F29:19 BND BND EOR
%   N15:30/1  FIC212_AM  "FIC-21-2 Feed Flow No-2 Auto/Manual Mode 0 = Auto 1 = Manual" %
%   F29:18  FIC212_OUT_FP  "FIC-21-2 Output Value (For HMI Display)" %
%   N15:42  FIC212_OMIN  "FIC-21-2 Feed Flow No-2 Output Minimum" %
%   N15:41  FIC212_OMAX  "FIC-21-2 Feed Flow No-2 Output Maximum" %
%   N24:20  PID_MIN  "PID Statement Minimum Value" %
%   N24:21  PID_MAX  "PID Statement Maximum Value" %
%   N18:2  FIC212_OUT1  "FIC-21-2 Feed Flow No-2 PID Output Value" %
%   F29:140  SIC212_MIN  "SIC-21-2 PU-21-2 Feed Pump No-2 Speed 0% Value (For HMI Display)" %
%   F29:144  SIC212_MAX  "SIC-21-2 PU-21-2 Feed Pump No-2 Freq at 100% Value (For HMI Display)" %
%   F29:19  FIC212_SP_FP  "FIC-21-2 Setpoint Value (For HMI Display)" %
%   N15:32  FIC212_SP  "FIC-21-2 Feed Flow No-2 SetPoint" %
%   N15:44  FIC212_PV  "FIC-21-2 Feed Flow No-2 Scaled Process Variable" %
%   F29:15  FIC212_PV_FP  "FIC-21-2 PV Value (For HMI Display)" %

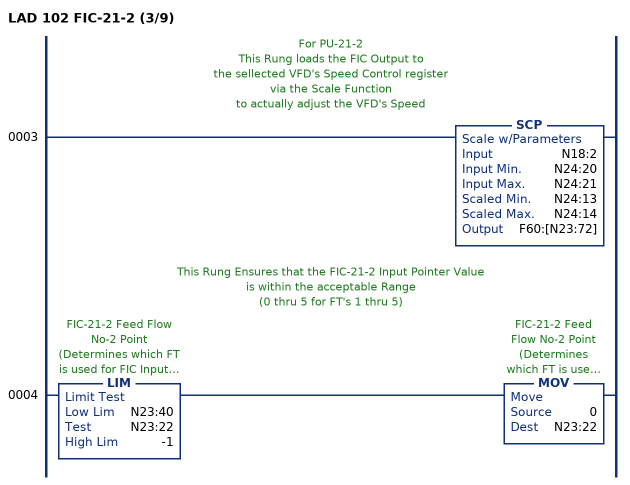
% Rung: 3 %
% For PU-21-2
% This Rung loads the FIC Output to
% the sellected VFD's Speed Control register
% via the Scale Function
% to actually adjust the VFD's Speed %
SOR SCP N18:2 N24:20 N24:21 N24:13 N24:14 F60:[N23:72] EOR
%   N18:2  FIC212_OUT1  "FIC-21-2 Feed Flow No-2 PID Output Value" %
%   N24:20  PID_MIN  "PID Statement Minimum Value" %
%   N24:21  PID_MAX  "PID Statement Maximum Value" %
%   N24:13  AO_MIN_OE4  "Analog Output Minimum Value Generates 4 mA DC (To OE4 AO Module)" %
%   N24:14  AO_MAX_OE4  "Analog Output Maximum Value Generates 20 mA DC (To OE4 AO Module)" %
%   N23:72  FIC212_OUT_PTR  "FIC-21-2 Feed Flow No-2 Output Pointer Determines which VFD is controled by FIC" %
% Rung: 4 %
% This Rung Ensures that the FIC-21-2 Input Pointer Value
% is within the acceptable Range
% (0 thru 5 for FT's 1 thru 5) %
SOR LIM N23:40 N23:22 -1 MOV 0 N23:22 EOR
%   N23:40  MAX_FT_ALLOWED_1  "Maximum Number of FTs Available Plus 1" %
%   N23:22  FIC212_IN_PTR  "FIC-21-2 Feed Flow No-2 Point (Determines which FT is used for FIC Input)" %

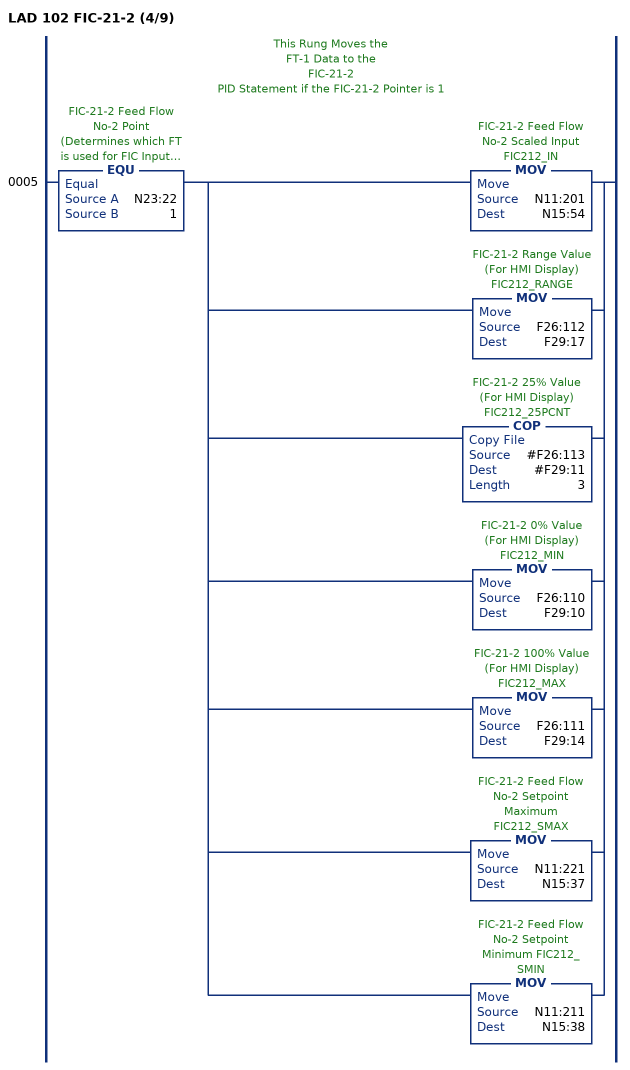
% Rung: 5 %
% This Rung Moves the
% FT-1 Data to the
% FIC-21-2
%  PID Statement if the FIC-21-2 Pointer is 1 %
SOR EQU N23:22 1 BST MOV N11:201 N15:54 NXB MOV F26:112 F29:17 NXB COP #F26:113 #F29:11 3 NXB MOV F26:110 F29:10 NXB MOV F26:111 F29:14 NXB MOV N11:221 N15:37 NXB MOV N11:211 N15:38 BND EOR
%   N23:22  FIC212_IN_PTR  "FIC-21-2 Feed Flow No-2 Point (Determines which FT is used for FIC Input)" %
%   N11:201  FT01_PID_IN  "FT-1 Flow Transmitter No-1 PID Statement Input Value" %
%   N15:54  FIC212_IN  "FIC-21-2 Feed Flow No-2 Scaled Input" %
%   F26:112  FT01_RANGE  "FT-1 Range Value (Max-Min)" %
%   F29:17  FIC212_RANGE  "FIC-21-2 Range Value (For HMI Display)" %
%   F26:113  FT01_25PCNT_VALUE  "FT-1 25% Range Value For HMI Display" %
%   F29:11  FIC212_25PCNT  "FIC-21-2 25% Value (For HMI Display)" %
%   F26:110  FT01_MIN  "FT-1 Minimum Value" %
%   F29:10  FIC212_MIN  "FIC-21-2 0% Value (For HMI Display)" %
%   F26:111  FT01_MAX  "FT-1 Maximum Value" %
%   F29:14  FIC212_MAX  "FIC-21-2 100% Value (For HMI Display)" %
%   N11:221  FT01_PID_MAX  "FT-1 Flow Transmitter No-1 PID Statement Maximum Input Value" %
%   N15:37  FIC212_SMAX  "FIC-21-2 Feed Flow No-2 Setpoint Maximum" %
%   N11:211  FT01_PID_MIN  "FT-1 Flow Transmitter No-1 PID Statement Minimum Input Value" %
%   N15:38  FIC212_SMIN  "FIC-21-2 Feed Flow No-2 Setpoint Minimum" %

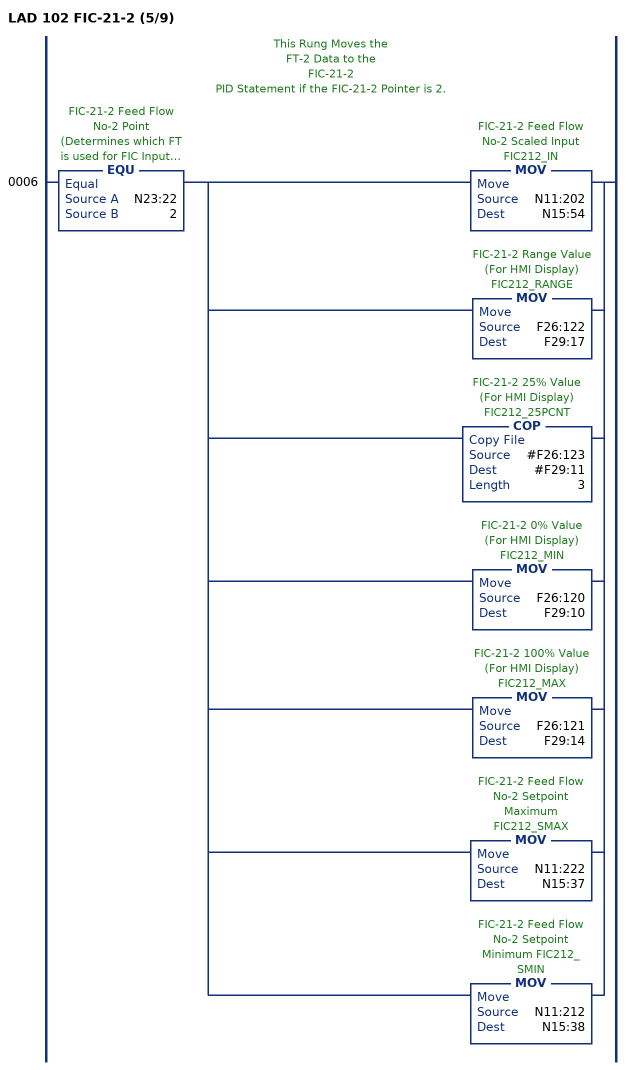
% Rung: 6 %
% This Rung Moves the
% FT-2 Data to the
% FIC-21-2
% PID Statement if the FIC-21-2 Pointer is 2. %
SOR EQU N23:22 2 BST MOV N11:202 N15:54 NXB MOV F26:122 F29:17 NXB COP #F26:123 #F29:11 3 NXB MOV F26:120 F29:10 NXB MOV F26:121 F29:14 NXB MOV N11:222 N15:37 NXB MOV N11:212 N15:38 BND EOR
%   N23:22  FIC212_IN_PTR  "FIC-21-2 Feed Flow No-2 Point (Determines which FT is used for FIC Input)" %
%   N11:202  FT02_PID_IN  "FT-2 Flow Transmitter No-2 PID Statement Input Value" %
%   N15:54  FIC212_IN  "FIC-21-2 Feed Flow No-2 Scaled Input" %
%   F26:122  FT02_RANGE  "FT-2 Range Value (Max-Min)" %
%   F29:17  FIC212_RANGE  "FIC-21-2 Range Value (For HMI Display)" %
%   F26:123  FT02_25PCNT_VALUE  "FT-2 25% Range Value For HMI Display" %
%   F29:11  FIC212_25PCNT  "FIC-21-2 25% Value (For HMI Display)" %
%   F26:120  FT02_MIN  "FT-2 Minimum Value" %
%   F29:10  FIC212_MIN  "FIC-21-2 0% Value (For HMI Display)" %
%   F26:121  FT02_MAX  "FT-2 Maximum Value" %
%   F29:14  FIC212_MAX  "FIC-21-2 100% Value (For HMI Display)" %
%   N11:222  FT02_PID_MAX  "FT-2 Flow Transmitter No-2 PID Statement Maximum Input Value" %
%   N15:37  FIC212_SMAX  "FIC-21-2 Feed Flow No-2 Setpoint Maximum" %
%   N11:212  FT02_PID_MIN  "FT-2 Flow Transmitter No-2 PID Statement Minimum Input Value" %
%   N15:38  FIC212_SMIN  "FIC-21-2 Feed Flow No-2 Setpoint Minimum" %

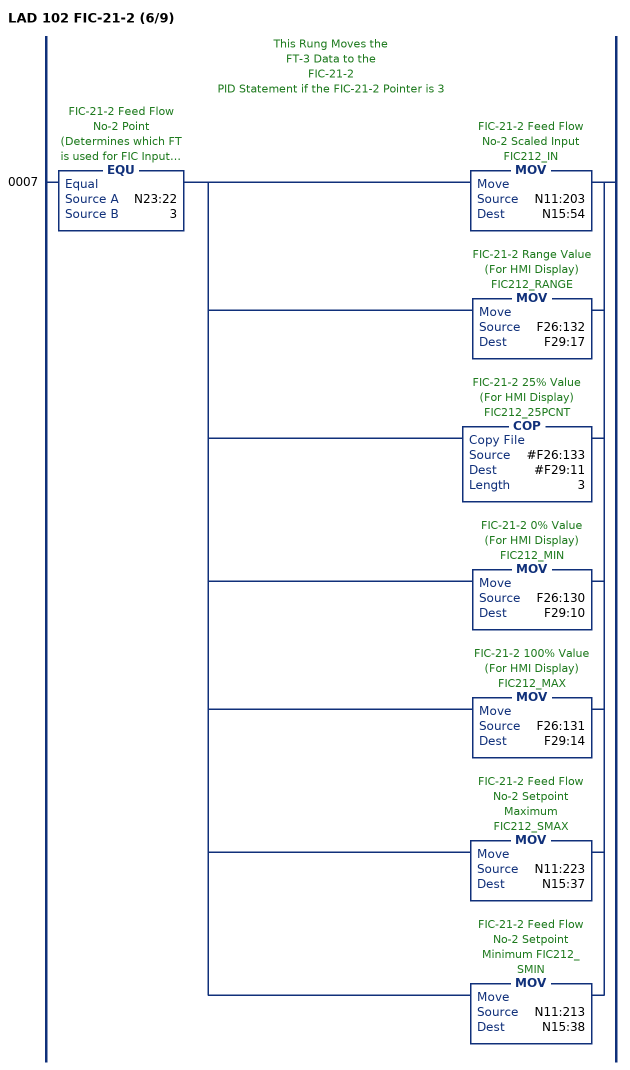
% Rung: 7 %
% This Rung Moves the
% FT-3 Data to the
% FIC-21-2
% PID Statement if the FIC-21-2 Pointer is 3 %
SOR EQU N23:22 3 BST MOV N11:203 N15:54 NXB MOV F26:132 F29:17 NXB COP #F26:133 #F29:11 3 NXB MOV F26:130 F29:10 NXB MOV F26:131 F29:14 NXB MOV N11:223 N15:37 NXB MOV N11:213 N15:38 BND EOR
%   N23:22  FIC212_IN_PTR  "FIC-21-2 Feed Flow No-2 Point (Determines which FT is used for FIC Input)" %
%   N11:203  FT03_PID_IN  "FT-3 Flow Transmitter No-3 PID Statement Input Value" %
%   N15:54  FIC212_IN  "FIC-21-2 Feed Flow No-2 Scaled Input" %
%   F26:132  FT03_RANGE  "FT-3 Range Value (Max-Min)" %
%   F29:17  FIC212_RANGE  "FIC-21-2 Range Value (For HMI Display)" %
%   F26:133  FT03_25PCNT_VALUE  "FT-3 25% Range Value For HMI Display" %
%   F29:11  FIC212_25PCNT  "FIC-21-2 25% Value (For HMI Display)" %
%   F26:130  FT03_MIN  "FT-3 Minimum Value" %
%   F29:10  FIC212_MIN  "FIC-21-2 0% Value (For HMI Display)" %
%   F26:131  FT03_MAX  "FT-3 Maximum Value" %
%   F29:14  FIC212_MAX  "FIC-21-2 100% Value (For HMI Display)" %
%   N11:223  FT03_PID_MAX  "FT-3 Flow Transmitter No-3 PID Statement Maximum Input Value" %
%   N15:37  FIC212_SMAX  "FIC-21-2 Feed Flow No-2 Setpoint Maximum" %
%   N11:213  FT03_PID_MIN  "FT-3 Flow Transmitter No-3 PID Statement Minimum Input Value" %
%   N15:38  FIC212_SMIN  "FIC-21-2 Feed Flow No-2 Setpoint Minimum" %

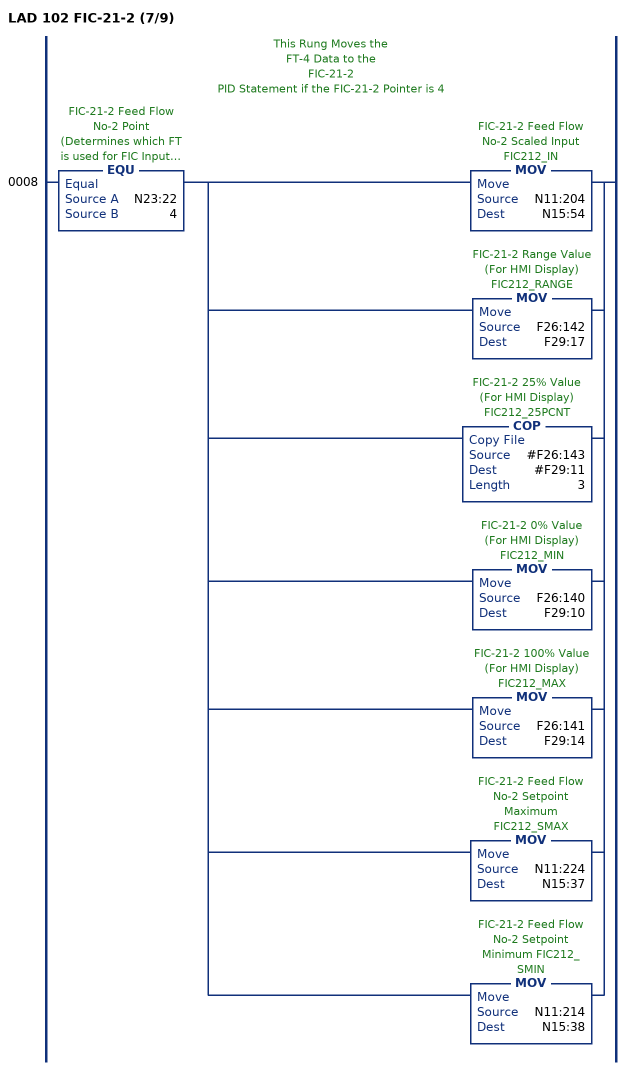
% Rung: 8 %
% This Rung Moves the
% FT-4 Data to the
% FIC-21-2
% PID Statement if the FIC-21-2 Pointer is 4 %
SOR EQU N23:22 4 BST MOV N11:204 N15:54 NXB MOV F26:142 F29:17 NXB COP #F26:143 #F29:11 3 NXB MOV F26:140 F29:10 NXB MOV F26:141 F29:14 NXB MOV N11:224 N15:37 NXB MOV N11:214 N15:38 BND EOR
%   N23:22  FIC212_IN_PTR  "FIC-21-2 Feed Flow No-2 Point (Determines which FT is used for FIC Input)" %
%   N11:204  FT04_PID_IN  "FT-4 Flow Transmitter No-4 PID Statement Input Value" %
%   N15:54  FIC212_IN  "FIC-21-2 Feed Flow No-2 Scaled Input" %
%   F26:142  FT04_RANGE  "FT-4 Range Value (Max-Min)" %
%   F29:17  FIC212_RANGE  "FIC-21-2 Range Value (For HMI Display)" %
%   F26:143  FT04_25PCNT_VALUE  "FT-4 25% Range Value For HMI Display" %
%   F29:11  FIC212_25PCNT  "FIC-21-2 25% Value (For HMI Display)" %
%   F26:140  FT04_MIN  "FT-4 Minimum Value" %
%   F29:10  FIC212_MIN  "FIC-21-2 0% Value (For HMI Display)" %
%   F26:141  FT04_MAX  "FT-4 Maximum Value" %
%   F29:14  FIC212_MAX  "FIC-21-2 100% Value (For HMI Display)" %
%   N11:224  FT04_PID_MAX  "FT-4 Flow Transmitter No-4 PID Statement Maximum Input Value" %
%   N15:37  FIC212_SMAX  "FIC-21-2 Feed Flow No-2 Setpoint Maximum" %
%   N11:214  FT04_PID_MIN  "FT-4 Flow Transmitter No-4 PID Statement Minimum Input Value" %
%   N15:38  FIC212_SMIN  "FIC-21-2 Feed Flow No-2 Setpoint Minimum" %

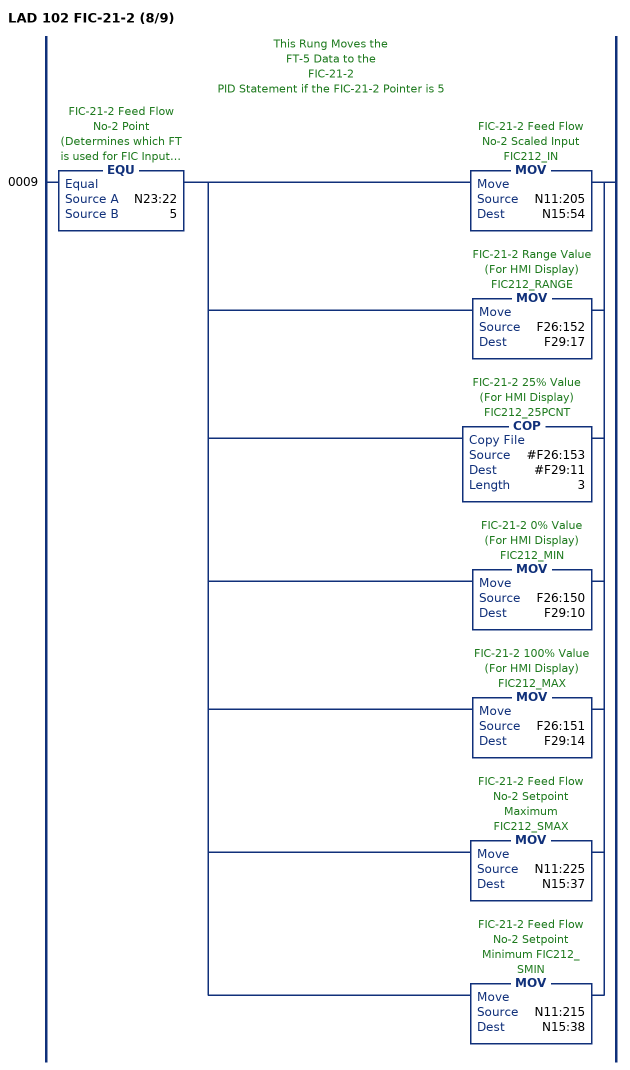
% Rung: 9 %
% This Rung Moves the
% FT-5 Data to the
% FIC-21-2
% PID Statement if the FIC-21-2 Pointer is 5 %
SOR EQU N23:22 5 BST MOV N11:205 N15:54 NXB MOV F26:152 F29:17 NXB COP #F26:153 #F29:11 3 NXB MOV F26:150 F29:10 NXB MOV F26:151 F29:14 NXB MOV N11:225 N15:37 NXB MOV N11:215 N15:38 BND EOR
%   N23:22  FIC212_IN_PTR  "FIC-21-2 Feed Flow No-2 Point (Determines which FT is used for FIC Input)" %
%   N11:205  FT05_PID_IN  "FT-5 Flow Transmitter No-5 PID Statement Input Value" %
%   N15:54  FIC212_IN  "FIC-21-2 Feed Flow No-2 Scaled Input" %
%   F26:152  FT05_RANGE  "FT-5 Range Value (Max-Min)" %
%   F29:17  FIC212_RANGE  "FIC-21-2 Range Value (For HMI Display)" %
%   F26:153  FT05_25PCNT_VALUE  "FT-5 25% Range Value For HMI Display" %
%   F29:11  FIC212_25PCNT  "FIC-21-2 25% Value (For HMI Display)" %
%   F26:150  FT05_MIN  "FT-5 Minimum Value" %
%   F29:10  FIC212_MIN  "FIC-21-2 0% Value (For HMI Display)" %
%   F26:151  FT05_MAX  "FT-5 Maximum Value" %
%   F29:14  FIC212_MAX  "FIC-21-2 100% Value (For HMI Display)" %
%   N11:225  FT05_PID_MAX  "FT-5 Flow Transmitter No-5 PID Statement Maximum Input Value" %
%   N15:37  FIC212_SMAX  "FIC-21-2 Feed Flow No-2 Setpoint Maximum" %
%   N11:215  FT05_PID_MIN  "FT-5 Flow Transmitter No-5 PID Statement Minimum Input Value" %
%   N15:38  FIC212_SMIN  "FIC-21-2 Feed Flow No-2 Setpoint Minimum" %

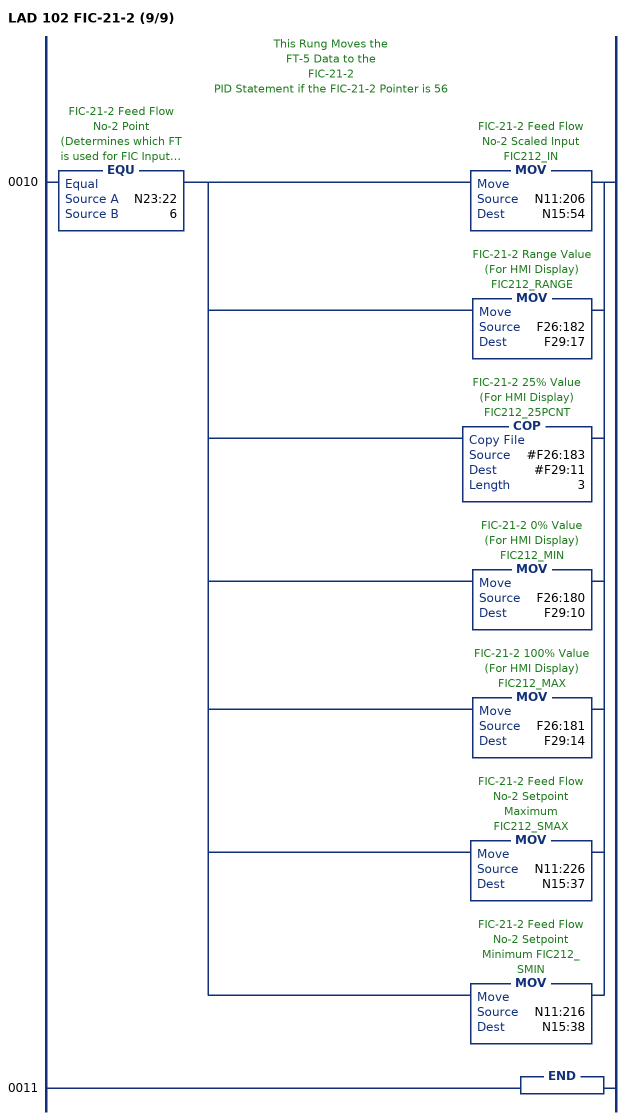
% Rung: 10 %
% This Rung Moves the
% FT-5 Data to the
% FIC-21-2
% PID Statement if the FIC-21-2 Pointer is 56 %
SOR EQU N23:22 6 BST MOV N11:206 N15:54 NXB MOV F26:182 F29:17 NXB COP #F26:183 #F29:11 3 NXB MOV F26:180 F29:10 NXB MOV F26:181 F29:14 NXB MOV N11:226 N15:37 NXB MOV N11:216 N15:38 BND EOR
%   N23:22  FIC212_IN_PTR  "FIC-21-2 Feed Flow No-2 Point (Determines which FT is used for FIC Input)" %
%   N11:206  FT06_PID_IN  "FT-6 Flow Transmitter No-6 PID Statement Input Value" %
%   N15:54  FIC212_IN  "FIC-21-2 Feed Flow No-2 Scaled Input" %
%   F26:182  FT06_RANGE  "FT-6 Range Value (Max-Min)" %
%   F29:17  FIC212_RANGE  "FIC-21-2 Range Value (For HMI Display)" %
%   F26:183  FT06_25PCNT_VALUE  "FT-6 25% Range Value For HMI Display" %
%   F29:11  FIC212_25PCNT  "FIC-21-2 25% Value (For HMI Display)" %
%   F26:180  FT06_MIN  "FT-6 Minimum Value" %
%   F29:10  FIC212_MIN  "FIC-21-2 0% Value (For HMI Display)" %
%   F26:181  FT06_MAX  "FT-6 Maximum Value" %
%   F29:14  FIC212_MAX  "FIC-21-2 100% Value (For HMI Display)" %
%   N11:226  FT06_PID_MAX  "FT-6 Flow Transmitter No-6 PID Statement Maximum Input Value" %
%   N15:37  FIC212_SMAX  "FIC-21-2 Feed Flow No-2 Setpoint Maximum" %
%   N11:216  FT06_PID_MIN  "FT-6 Flow Transmitter No-6 PID Statement Minimum Input Value" %
%   N15:38  FIC212_SMIN  "FIC-21-2 Feed Flow No-2 Setpoint Minimum" %
% Rung: 11 %
SOR END EOR

LADDER 103 "FIC-21-3"    % Feed Flow No-3 PID Controls %
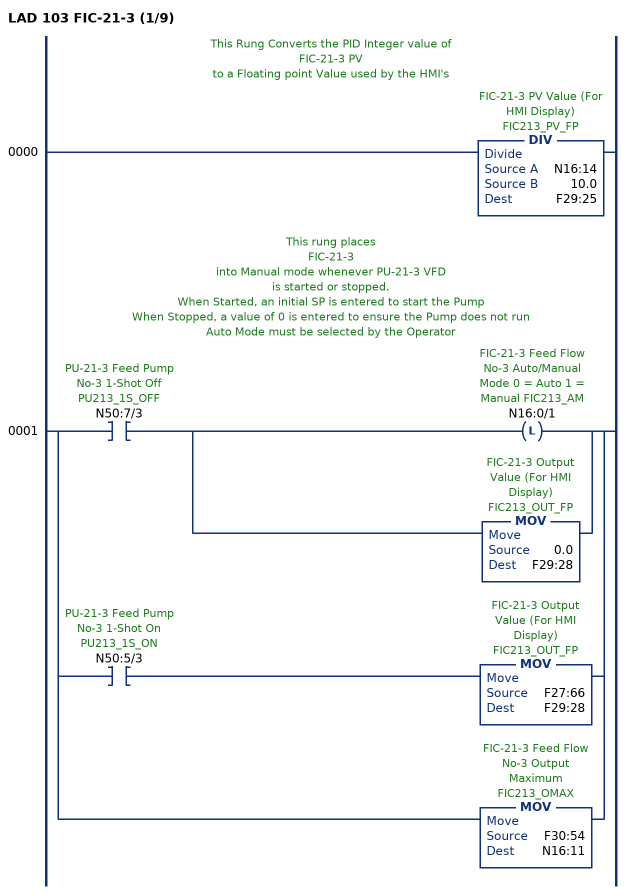
% Rung: 0 %
% This Rung Converts the PID Integer value of
% FIC-21-3 PV
% to a Floating point Value used by the HMI's %
SOR DIV N16:14 10.0 F29:25 EOR
%   N16:14  FIC213_PV  "FIC-21-3 Feed Flow No-3 Scaled Process Variable" %
%   F29:25  FIC213_PV_FP  "FIC-21-3 PV Value (For HMI Display)" %
% Rung: 1 %
% This rung places
% FIC-21-3
% into Manual mode whenever PU-21-3 VFD
% is started or stopped.
% When Started, an initial SP is entered to start the Pump
% When Stopped, a value of 0 is entered to ensure the Pump does not run
% Auto Mode must be selected by the Operator %
SOR BST XIC N50:7/3 BST OTL N16:0/1 NXB MOV 0.0 F29:28 BND NXB XIC N50:5/3 MOV F27:66 F29:28 NXB MOV F30:54 N16:11 BND EOR
%   N50:7/3  PU213_1S_OFF  "PU-21-3 Feed Pump No-3 1-Shot Off" %
%   N16:0/1  FIC213_AM  "FIC-21-3 Feed Flow No-3 Auto/Manual Mode 0 = Auto 1 = Manual" %
%   F29:28  FIC213_OUT_FP  "FIC-21-3 Output Value (For HMI Display)" %
%   N50:5/3  PU213_1S_ON  "PU-21-3 Feed Pump No-3 1-Shot On" %
%   F27:66  SIC213_INIT_SP  "SIC-21-3 Initial Speed Setpoint (Hz)" %
%   F30:54  SIC213_MAX  "SIC-21-3 PU-21-3 Feed Pump No-3 Freq at 100% Value (For HMI Display)" %
%   N16:11  FIC213_OMAX  "FIC-21-3 Feed Flow No-3 Output Maximum" %

